REGION Network 2: Yeşil lamba
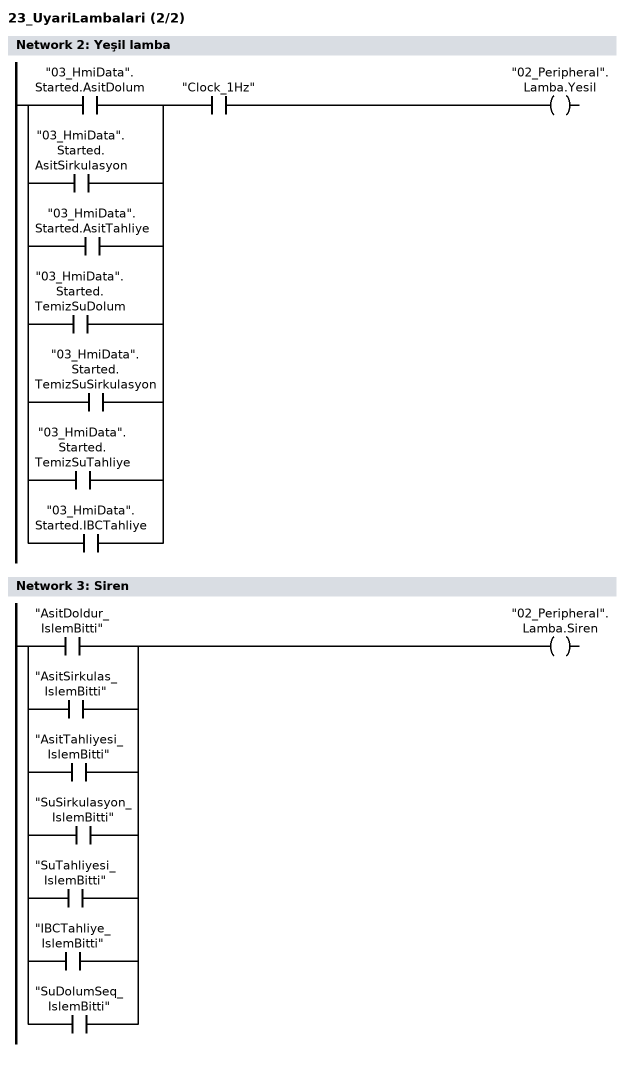
   RUNG wire#powerrail
      Contact( "03_HmiData".Started.AsitDolum )
      wire#w1
      Contact( "Clock_1Hz" )
      Coil( "02_Peripheral".Lamba.Yesil )
   END_RUNG
   RUNG wire#powerrail
      Contact( "03_HmiData".Started.AsitSirkulasyon )
   END_RUNG wire#w1
   RUNG wire#powerrail
      Contact( "03_HmiData".Started.AsitTahliye )
   END_RUNG wire#w1
   RUNG wire#powerrail
      Contact( "03_HmiData".Started.TemizSuDolum )
   END_RUNG wire#w1
   RUNG wire#powerrail
      Contact( "03_HmiData".Started.TemizSuSirkulasyon )
   END_RUNG wire#w1
   RUNG wire#powerrail
      Contact( "03_HmiData".Started.TemizSuTahliye )
   END_RUNG wire#w1
   RUNG wire#powerrail
      Contact( "03_HmiData".Started.IBCTahliye )
   END_RUNG wire#w1
   // the same network as SCL:
   "02_Peripheral".Lamba.Yesil := ("03_HmiData".Started.AsitDolum OR "03_HmiData".Started.AsitSirkulasyon OR "03_HmiData".Started.AsitTahliye OR "03_HmiData".Started.TemizSuDolum OR "03_HmiData".Started.TemizSuSirkulasyon OR "03_HmiData".Started.TemizSuTahliye OR "03_HmiData".Started.IBCTahliye) AND "Clock_1Hz";
END_REGION

REGION Network 3: Siren
   RUNG wire#powerrail
      Contact( "AsitDoldur_IslemBitti" )
      wire#w1
      Coil( "02_Peripheral".Lamba.Siren )
   END_RUNG
   RUNG wire#powerrail
      Contact( "AsitSirkulas_IslemBitti" )
   END_RUNG wire#w1
   RUNG wire#powerrail
      Contact( "AsitTahliyesi_IslemBitti" )
   END_RUNG wire#w1
   RUNG wire#powerrail
      Contact( "SuSirkulasyon_IslemBitti" )
   END_RUNG wire#w1
   RUNG wire#powerrail
      Contact( "SuTahliyesi_IslemBitti" )
   END_RUNG wire#w1
   RUNG wire#powerrail
      Contact( "IBCTahliye_IslemBitti" )
   END_RUNG wire#w1
   RUNG wire#powerrail
      Contact( "SuDolumSeq_IslemBitti" )
   END_RUNG wire#w1
   // the same network as SCL:
   "02_Peripheral".Lamba.Siren := "AsitDoldur_IslemBitti" OR "AsitSirkulas_IslemBitti" OR "AsitTahliyesi_IslemBitti" OR "SuSirkulasyon_IslemBitti" OR "SuTahliyesi_IslemBitti" OR "IBCTahliye_IslemBitti" OR "SuDolumSeq_IslemBitti";
END_REGION
END_FUNCTION

FUNCTION "14_SuDolumuSeq" : Void   // FC10, LAD
{ S7_Optimized_Access := 'TRUE' }
VERSION : 0.1
BEGIN

REGION Network 1
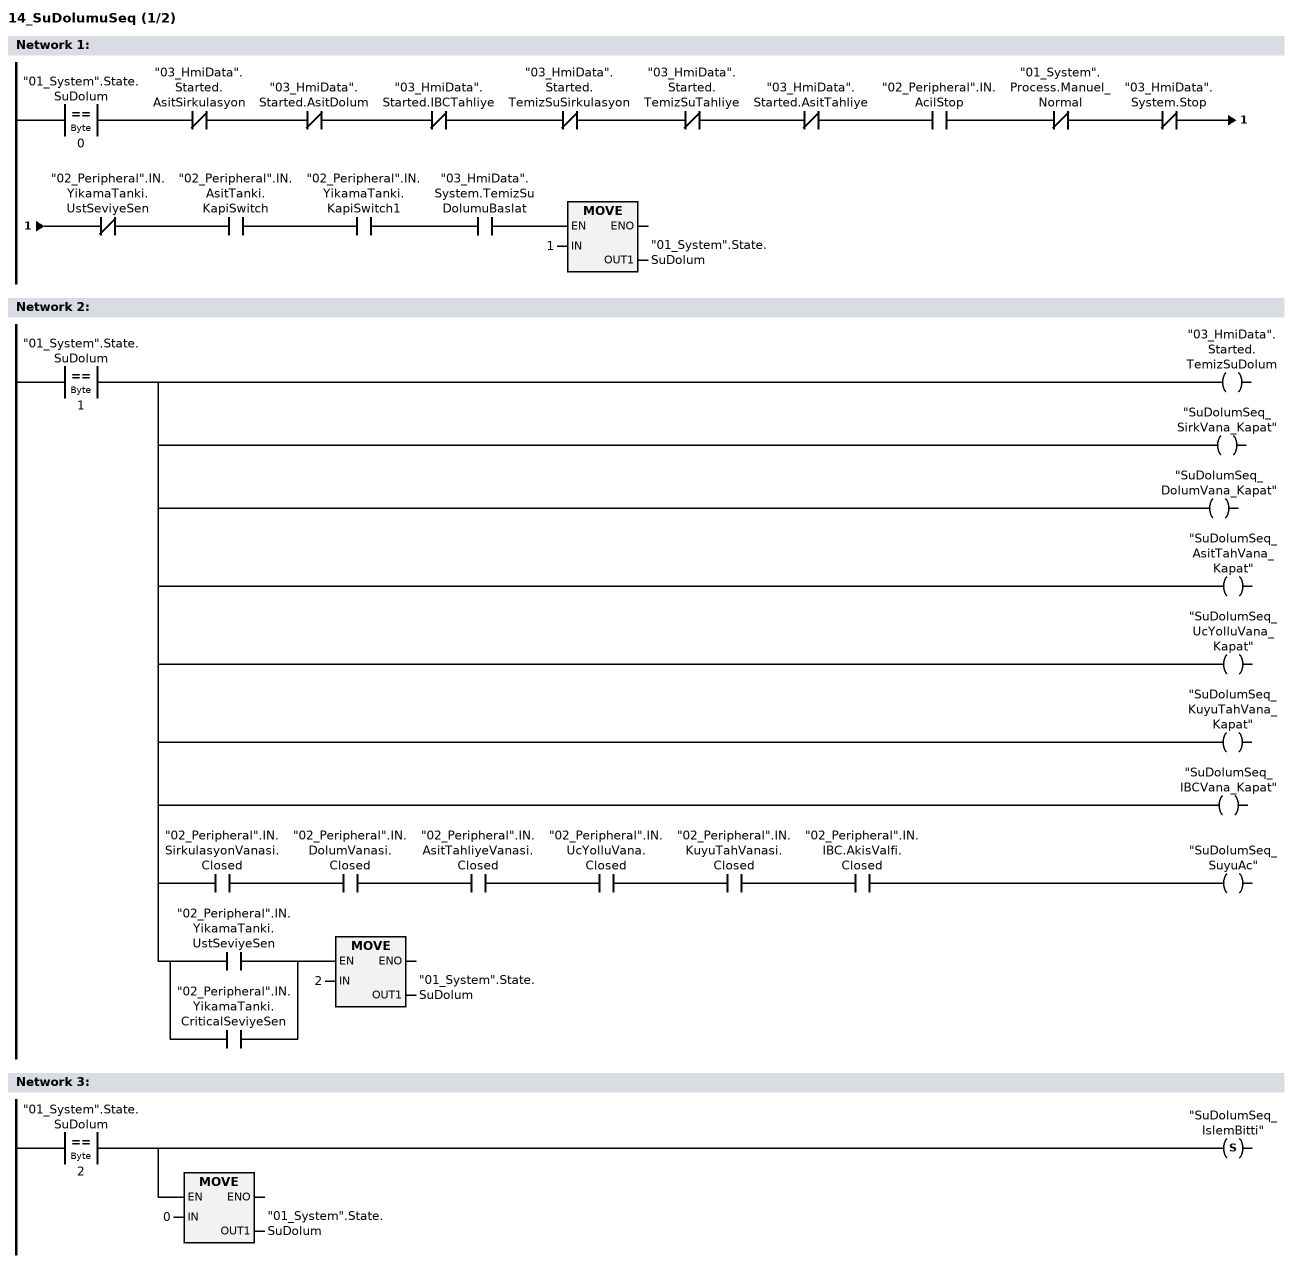
   RUNG wire#powerrail
      { S7_Templates := "SrcType := Byte" } EQ_Contact(in1 := "01_System".State.SuDolum, in2 := 0)
      I_Contact( "03_HmiData".Started.AsitSirkulasyon )
      I_Contact( "03_HmiData".Started.AsitDolum )
      I_Contact( "03_HmiData".Started.IBCTahliye )
      I_Contact( "03_HmiData".Started.TemizSuSirkulasyon )
      I_Contact( "03_HmiData".Started.TemizSuTahliye )
      I_Contact( "03_HmiData".Started.AsitTahliye )
      Contact( "02_Peripheral".IN.AcilStop )
      I_Contact( "01_System".Process.Manuel_Normal )
      I_Contact( "03_HmiData".System.Stop )
      I_Contact( "02_Peripheral".IN.YikamaTanki.UstSeviyeSen )
      Contact( "02_Peripheral".IN.AsitTanki.KapiSwitch )
      Contact( "02_Peripheral".IN.YikamaTanki.KapiSwitch1 )
      Contact( "03_HmiData".System.TemizSuDolumuBaslat )
      Move(in := 1, out1 => "01_System".State.SuDolum)
   END_RUNG
   // the same network as SCL:
   IF ("01_System".State.SuDolum = 0) AND NOT "03_HmiData".Started.AsitSirkulasyon AND NOT "03_HmiData".Started.AsitDolum AND NOT "03_HmiData".Started.IBCTahliye AND NOT "03_HmiData".Started.TemizSuSirkulasyon AND NOT "03_HmiData".Started.TemizSuTahliye AND NOT "03_HmiData".Started.AsitTahliye AND "02_Peripheral".IN.AcilStop AND NOT "01_System".Process.Manuel_Normal AND NOT "03_HmiData".System.Stop AND NOT "02_Peripheral".IN.YikamaTanki.UstSeviyeSen AND "02_Peripheral".IN.AsitTanki.KapiSwitch AND "02_Peripheral".IN.YikamaTanki.KapiSwitch1 AND "03_HmiData".System.TemizSuDolumuBaslat THEN
       "01_System".State.SuDolum := 1;
   END_IF;
END_REGION

REGION Network 2
   RUNG wire#powerrail
      { S7_Templates := "SrcType := Byte" } EQ_Contact(in1 := "01_System".State.SuDolum, in2 := 1)
      wire#w1
      Coil( "03_HmiData".Started.TemizSuDolum )
   END_RUNG
   RUNG wire#w1
      Coil( "SuDolumSeq_SirkVana_Kapat" )
   END_RUNG
   RUNG wire#w1
      Coil( "SuDolumSeq_DolumVana_Kapat" )
   END_RUNG
   RUNG wire#w1
      Coil( "SuDolumSeq_AsitTahVana_Kapat" )
   END_RUNG
   RUNG wire#w1
      Coil( "SuDolumSeq_UcYolluVana_Kapat" )
   END_RUNG
   RUNG wire#w1
      Coil( "SuDolumSeq_KuyuTahVana_Kapat" )
   END_RUNG
   RUNG wire#w1
      Coil( "SuDolumSeq_IBCVana_Kapat" )
   END_RUNG
   RUNG wire#w1
      Contact( "02_Peripheral".IN.SirkulasyonVanasi.Closed )
      Contact( "02_Peripheral".IN.DolumVanasi.Closed )
      Contact( "02_Peripheral".IN.AsitTahliyeVanasi.Closed )
      Contact( "02_Peripheral".IN.UcYolluVana.Closed )
      Contact( "02_Peripheral".IN.KuyuTahVanasi.Closed )
      Contact( "02_Peripheral".IN.IBC.AkisValfi.Closed )
      Coil( "SuDolumSeq_SuyuAc" )
   END_RUNG
   RUNG wire#w1
      Contact( "02_Peripheral".IN.YikamaTanki.UstSeviyeSen )
      wire#w2
      Move(in := 2, out1 => "01_System".State.SuDolum)
   END_RUNG
   RUNG wire#w1
      Contact( "02_Peripheral".IN.YikamaTanki.CriticalSeviyeSen )
   END_RUNG wire#w2
   // the same network as SCL:
   "03_HmiData".Started.TemizSuDolum := "01_System".State.SuDolum = 1;
   "SuDolumSeq_SirkVana_Kapat" := "03_HmiData".Started.TemizSuDolum;
   "SuDolumSeq_DolumVana_Kapat" := "03_HmiData".Started.TemizSuDolum;
   "SuDolumSeq_AsitTahVana_Kapat" := "03_HmiData".Started.TemizSuDolum;
   "SuDolumSeq_UcYolluVana_Kapat" := "03_HmiData".Started.TemizSuDolum;
   "SuDolumSeq_KuyuTahVana_Kapat" := "03_HmiData".Started.TemizSuDolum;
   "SuDolumSeq_IBCVana_Kapat" := "03_HmiData".Started.TemizSuDolum;
   "SuDolumSeq_SuyuAc" := "03_HmiData".Started.TemizSuDolum AND "02_Peripheral".IN.SirkulasyonVanasi.Closed AND "02_Peripheral".IN.DolumVanasi.Closed AND "02_Peripheral".IN.AsitTahliyeVanasi.Closed AND "02_Peripheral".IN.UcYolluVana.Closed AND "02_Peripheral".IN.KuyuTahVanasi.Closed AND "02_Peripheral".IN.IBC.AkisValfi.Closed;
   IF "03_HmiData".Started.TemizSuDolum AND ("02_Peripheral".IN.YikamaTanki.UstSeviyeSen OR "02_Peripheral".IN.YikamaTanki.CriticalSeviyeSen) THEN
       "01_System".State.SuDolum := 2;
   END_IF;
END_REGION

REGION Network 3
   RUNG wire#powerrail
      { S7_Templates := "SrcType := Byte" } EQ_Contact(in1 := "01_System".State.SuDolum, in2 := 2)
      wire#w1
      S_Coil( "SuDolumSeq_IslemBitti" )
   END_RUNG
   RUNG wire#w1
      Move(in := 0, out1 => "01_System".State.SuDolum)
   END_RUNG
   // the same network as SCL:
   IF "01_System".State.SuDolum = 2 THEN
       "SuDolumSeq_IslemBitti" := TRUE;
       "01_System".State.SuDolum := 0;
   END_IF;
END_REGION

REGION Network 4
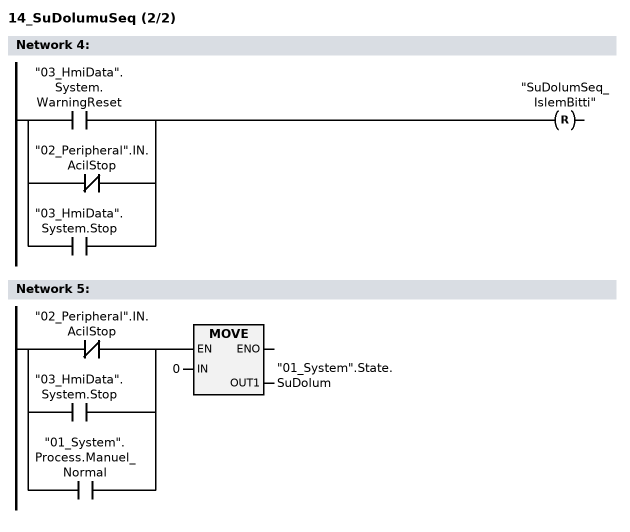
   RUNG wire#powerrail
      Contact( "03_HmiData".System.WarningReset )
      wire#w1
      R_Coil( "SuDolumSeq_IslemBitti" )
   END_RUNG
   RUNG wire#powerrail
      I_Contact( "02_Peripheral".IN.AcilStop )
   END_RUNG wire#w1
   RUNG wire#powerrail
      Contact( "03_HmiData".System.Stop )
   END_RUNG wire#w1
   // the same network as SCL:
   IF "03_HmiData".System.WarningReset OR NOT "02_Peripheral".IN.AcilStop OR "03_HmiData".System.Stop THEN
       "SuDolumSeq_IslemBitti" := FALSE;
   END_IF;
END_REGION

REGION Network 5
   RUNG wire#powerrail
      I_Contact( "02_Peripheral".IN.AcilStop )
      wire#w1
      Move(in := 0, out1 => "01_System".State.SuDolum)
   END_RUNG
   RUNG wire#powerrail
      Contact( "03_HmiData".System.Stop )
   END_RUNG wire#w1
   RUNG wire#powerrail
      Contact( "01_System".Process.Manuel_Normal )
   END_RUNG wire#w1
   // the same network as SCL:
   IF NOT "02_Peripheral".IN.AcilStop OR "03_HmiData".System.Stop OR "01_System".Process.Manuel_Normal THEN
       "01_System".State.SuDolum := 0;
   END_IF;
END_REGION
END_FUNCTION

ORGANIZATION_BLOCK "Main"   // OB1, FBD, ProgramCycle
TITLE = "Main Program Sweep (Cycle)"
{ S7_Optimized_Access := 'TRUE' }
VERSION : 0.1
   VAR_INPUT
      Initial_Call : Bool;   // Initial call of this OB
      Remanence : Bool;   // =True, if remanent data are available
   END_VAR
BEGIN

REGION Network 1: Manuel
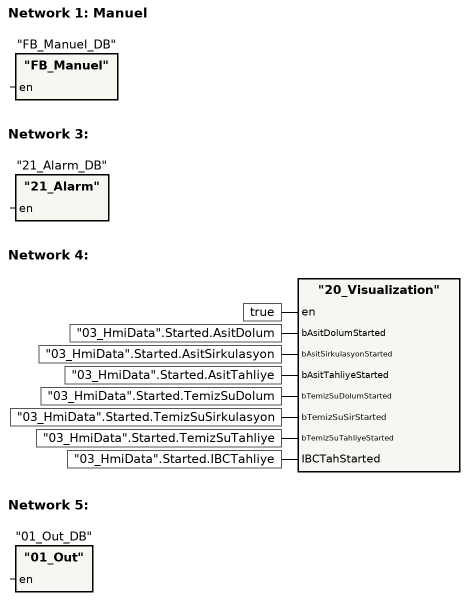
   "FB_Manuel_DB"();   // "FB_Manuel"
END_REGION

REGION Network 2 (SCL): Otomatik sekanslar
   "11_AsitDolumSeq"();
   "12_AsitSirkulasyonSeq"();
   "13_AsitTahliyeSeq"();
   "14_SuDolumuSeq"();
   "15_SuSirkulasyonSeq"();
   "16_SuTahliyeSeq"();
   "17_IBCTahliyeSeq"();

   "22_Peripheral"();
   "23_UyariLambalari"();

   "Always_On" := true;
END_REGION

REGION Network 3
   "21_Alarm_DB"();   // "21_Alarm"
END_REGION

REGION Network 4
   IF true THEN
       "20_Visualization"(bAsitDolumStarted := "03_HmiData".Started.AsitDolum,
                          bAsitSirkulasyonStarted := "03_HmiData".Started.AsitSirkulasyon,
                          bAsitTahliyeStarted := "03_HmiData".Started.AsitTahliye,
                          bTemizSuDolumStarted := "03_HmiData".Started.TemizSuDolum,
                          bTemizSuSirStarted := "03_HmiData".Started.TemizSuSirkulasyon,
                          bTemizSuTahliyeStarted := "03_HmiData".Started.TemizSuTahliye,
                          IBCTahStarted := "03_HmiData".Started.IBCTahliye);
   END_IF;
END_REGION

REGION Network 5
   "01_Out_DB"();   // "01_Out"
END_REGION
END_ORGANIZATION_BLOCK

// folder: OB

ORGANIZATION_BLOCK "Time error interrupt"   // OB80, LAD, TimeErrorInterrupt
{ S7_Optimized_Access := 'TRUE' }
VERSION : 0.1
   VAR_INPUT
      Fault_ID : Byte;   // Fault identifier
      Csg_OBnr : OB_Any;   // Number of OB causing the error
      Csg_Prio : UInt;   // Priority of OB causing the error
   END_VAR
BEGIN
END_ORGANIZATION_BLOCK

ORGANIZATION_BLOCK "Pull or plug of modules"   // OB83, LAD, PullPlug
{ S7_Optimized_Access := 'TRUE' }
VERSION : 0.1
   VAR_INPUT
      LADDR : Hw_Io;   // Hardware identifier
      Event_Class : Byte;   // 16#38/39: module inserted, removed
      Fault_ID : Byte;   // Fault identifier
   END_VAR
BEGIN
END_ORGANIZATION_BLOCK

ORGANIZATION_BLOCK "Rack or station failure"   // OB86, LAD, RackStationFailure
{ S7_Optimized_Access := 'TRUE' }
VERSION : 0.1
   VAR_INPUT
      LADDR : Hw_Device;   // Hardware identifier
      Event_Class : Byte;   // Event class
      Fault_ID : Byte;   // Fault identifier
   END_VAR
BEGIN
END_ORGANIZATION_BLOCK

ORGANIZATION_BLOCK "Startup"   // OB100, LAD, Startup
TITLE = "Complete Restart"
{ S7_Optimized_Access := 'TRUE' }
VERSION : 0.1
   VAR_INPUT
      LostRetentive : Bool;   // True if retentive data are lost
      LostRTC : Bool;   // True if date and time are lost
   END_VAR
BEGIN

REGION Network 1
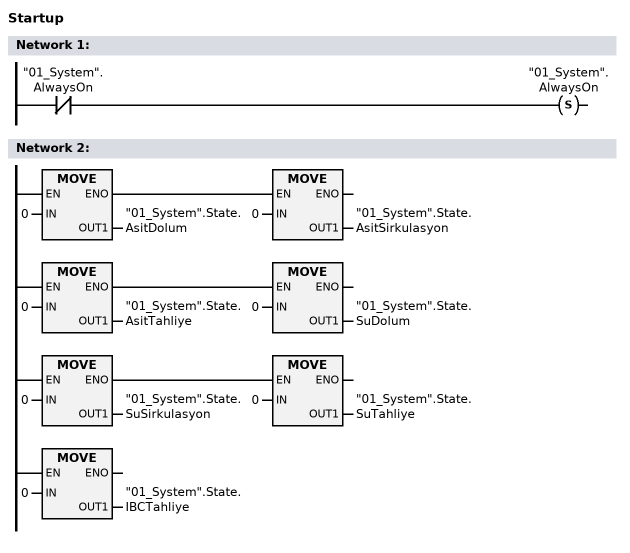
   RUNG wire#powerrail
      I_Contact( "01_System".AlwaysOn )
      S_Coil( "01_System".AlwaysOn )
   END_RUNG
   // the same network as SCL:
   IF NOT "01_System".AlwaysOn THEN "01_System".AlwaysOn := TRUE; END_IF;
END_REGION

REGION Network 2
   RUNG wire#powerrail
      Move(in := 0, out1 => "01_System".State.AsitDolum)
      Move(in := 0, out1 => "01_System".State.AsitSirkulasyon)
   END_RUNG
   RUNG wire#powerrail
      Move(in := 0, out1 => "01_System".State.AsitTahliye)
      Move(in := 0, out1 => "01_System".State.SuDolum)
   END_RUNG
   RUNG wire#powerrail
      Move(in := 0, out1 => "01_System".State.SuSirkulasyon)
      Move(in := 0, out1 => "01_System".State.SuTahliye)
   END_RUNG
   RUNG wire#powerrail
      Move(in := 0, out1 => "01_System".State.IBCTahliye)
   END_RUNG
   // the same network as SCL:
   "01_System".State.AsitDolum := 0;
   "01_System".State.AsitSirkulasyon := 0;
   "01_System".State.AsitTahliye := 0;
   "01_System".State.SuDolum := 0;
   "01_System".State.SuSirkulasyon := 0;
   "01_System".State.SuTahliye := 0;
   "01_System".State.IBCTahliye := 0;
END_REGION
END_ORGANIZATION_BLOCK

(* ===== HMI "HMI_RT_1" =====
system functions are stored by id; their names below are inferred from use
connection "HMI_Connection_1": ETHERNET, SMART_S7_1200_OMS

HMI tags "Default tag table"
   "01_System_SystemInfo" : String[50] = PLC "01_System".SystemInfo, 100 ms
   "TestInfo" : WString[254] AT %DB1.DBX0.0
   "01_System_Alarms" : Word = PLC "01_System".Alarms, 1 s
   "01_System_Process.Manuel_Normal" : Bool = PLC "01_System".Process.Manuel_Normal, 100 ms
   "02_Peripheral_OUT.KorKuyuPompasi" : Bool = PLC "02_Peripheral".OUT.KorKuyuPompasi, 500 ms
   "HmiAnaPompa_Run" : Bool = PLC HmiAnaPompa_Run AT %M2.4, 1 s
   "HmiIBCPopmpa_Run" : Bool = PLC HmiIBCPopmpa_Run AT %M2.5, 1 s
   "HmiKorKuyuPompa_Run" : Bool = PLC HmiKorKuyuPompa_Run AT %M10.5, 1 s
   "03_HmiData_SoDulumVanasi_Ac" : Bool = PLC "03_HmiData".SuDolumVanasi_Ac, 1 s
   "03_HmiData_SuDolumVanasi_Kapat" : Bool = PLC "03_HmiData".SuDolumVanasi_Kapat, 1 s
   "02_Peripheral_OUT.SuDolumVanasi" : Bool = PLC "02_Peripheral".OUT.SuDolumVanasi, 1 s

HMI tags "00_HMI"
   "03_HmiData_SurkilasyonVanasi_Ac" : Bool = PLC "03_HmiData".SurkilasyonVanasi_Ac, 100 ms
   "03_HmiData_SurkilasyonVanasi_Kapat" : Bool = PLC "03_HmiData".SurkilasyonVanasi_Kapat, 100 ms
   "03_HmiData_DolumVanasi_Ac" : Bool = PLC "03_HmiData".DolumVanasi_Ac, 100 ms
   "03_HmiData_DolumVanasi_Kapat" : Bool = PLC "03_HmiData".DolumVanasi_Kapat, 100 ms
   "03_HmiData_AsitTahliyeVanasi_Ac" : Bool = PLC "03_HmiData".AsitTahliyeVanasi_Ac, 100 ms
   "03_HmiData_AsitTahliyeVanasi_Kapat" : Bool = PLC "03_HmiData".AsitTahliyeVanasi_Kapat, 100 ms
   "03_HmiData_UcYolluVana_Ac" : Bool = PLC "03_HmiData".UcYolluVana_Ac, 100 ms
   "03_HmiData_UcYolluVana_Kapat" : Bool = PLC "03_HmiData".UcYolluVana_Kapat, 100 ms
   "03_HmiData_KuyuAktarimVanasi_Ac" : Bool = PLC "03_HmiData".KuyuAktarimVanasi_Ac, 100 ms
   "03_HmiData_KuyuAktarimVanasi_Kapat" : Bool = PLC "03_HmiData".KuyuAktarimVanasi_Kapat, 100 ms
   "03_HmiData_IBCVanasi_Ac" : Bool = PLC "03_HmiData".IBCVanasi_Ac, 100 ms
   "03_HmiData_IBCVanasi_Kapat" : Bool = PLC "03_HmiData".IBCVanasi_Kapat, 100 ms
   "03_HmiData_AnaPompa_Run" : Bool = PLC "03_HmiData".AnaPompa_Run, 100 ms
   "03_HmiData_AnaPompa_Stop" : Bool = PLC "03_HmiData".AnaPompa_Stop, 100 ms
   "03_HmiData_IBC_DiyaframPompa_Run" : Bool = PLC "03_HmiData".IBC_DiyaframPompa_Run, 100 ms
   "03_HmiData_IBC_DiyaframPompa_Stop" : Bool = PLC "03_HmiData".IBC_DiyaframPompa_Stop, 100 ms
   "03_HmiData_Started.AsitDolum" : Bool = PLC "03_HmiData".Started.AsitDolum, 1 s
   "03_HmiData_Started.AsitSirkulasyon" : Bool = PLC "03_HmiData".Started.AsitSirkulasyon, 1 s
   "03_HmiData_Started.AsitTahliye" : Bool = PLC "03_HmiData".Started.AsitTahliye, 1 s
   "03_HmiData_Started.IBCTahliye" : Bool = PLC "03_HmiData".Started.IBCTahliye, 1 s
   "03_HmiData_Started.TemizSuDolum" : Bool = PLC "03_HmiData".Started.TemizSuDolum, 1 s
   "03_HmiData_Started.TemizSuSirkulasyon" : Bool = PLC "03_HmiData".Started.TemizSuSirkulasyon, 1 s
   "03_HmiData_Started.TemizSuTahliye" : Bool = PLC "03_HmiData".Started.TemizSuTahliye, 1 s
   "03_HmiData_System.Stop" : Bool = PLC "03_HmiData".System.Stop, 1 s
   "03_HmiData_System.WarningReset" : Bool = PLC "03_HmiData".System.WarningReset, 1 s
   "03_HmiData_Visualization.ActTimer" : DInt = PLC "03_HmiData".Visualization.ActTimerMin, 1 s
   "03_HmiData_Visualization.TimerVisible" : Bool = PLC "03_HmiData".Visualization.TimerVisible, 1 s
   "03_HmiData_Visualization.Visibility.AsitDolum" : Bool = PLC "03_HmiData".Visualization.Visibility.AsitDolum, 1 s
   "03_HmiData_Visualization.Visibility.AsitSirkulasyon" : Bool = PLC "03_HmiData".Visualization.Visibility.AsitSirkulasyon, 1 s
   "03_HmiData_Visualization.Visibility.AsitTahliyesi" : Bool = PLC "03_HmiData".Visualization.Visibility.AsitTahliyesi, 1 s
   "03_HmiData_Visualization.Visibility.IBCTaliye" : Bool = PLC "03_HmiData".Visualization.Visibility.IBCTaliye, 1 s
   "03_HmiData_Visualization.Visibility.TemizSuDolum" : Bool = PLC "03_HmiData".Visualization.Visibility.TemizSuDolum, 1 s
   "03_HmiData_Visualization.Visibility.TemizSuSirkulasyon" : Bool = PLC "03_HmiData".Visualization.Visibility.TemizSuSirkulasyon, 1 s
   "03_HmiData_Visualization.Visibility.TemizSuTahliye" : Bool = PLC "03_HmiData".Visualization.Visibility.TemizSuTahliye, 1 s
   "03_HmiData_KorKuyuPompası_Run" : Bool = PLC "03_HmiData".KorKuyuPompası_Run, 500 ms
   "03_HmiData_KorKuyuPompası_Stop" : Bool = PLC "03_HmiData".KorKuyuPompası_Stop, 500 ms
   "03_HmiData_System.AsitDoldurBaslat" : Bool = PLC "03_HmiData".System.AsitDoldurBaslat, 500 ms
   "03_HmiData_System.AsitSirkulasyonBaslat" : Bool = PLC "03_HmiData".System.AsitSirkulasyonBaslat, 500 ms
   "03_HmiData_System.AsitTahliyesiBaslat" : Bool = PLC "03_HmiData".System.AsitTahliyesiBaslat, 500 ms
   "03_HmiData_System.IBCTahliyesiBaslat" : Bool = PLC "03_HmiData".System.IBCTahliyesiBaslat, 500 ms
   "03_HmiData_System.TemizSuDolumuBaslat" : Bool = PLC "03_HmiData".System.TemizSuDolumuBaslat, 500 ms
   "03_HmiData_System.TemizSuSirkulasyonuBaslat" : Bool = PLC "03_HmiData".System.TemizSuSirkulasyonuBaslat, 500 ms
   "03_HmiData_System.TemizSuTahliyesiBaslat" : Bool = PLC "03_HmiData".System.TemizSuTahliyesiBaslat, 500 ms
   "03_HmiData_TimerInterval.AsitSirkulasyon" : Time = PLC "03_HmiData".TimerInterval.AsitSirkulasyon, 500 ms
   "03_HmiData_TimerInterval.SuSirkulasyon" : Time = PLC "03_HmiData".TimerInterval.SuSirkulasyon, 500 ms
   "03_HmiData_Visualization.ActTimerSec" : DInt = PLC "03_HmiData".Visualization.ActTimerSec, 100 ms
   "03_HmiData_Visualization.Visibility.Manuel.AsitTahVanaAc" : Bool = PLC "03_HmiData".Visualization.Visibility.Manuel.AsitTahVanaAc, 1 s
   "03_HmiData_Visualization.Visibility.Manuel.AsitTahVanaKapat" : Bool = PLC "03_HmiData".Visualization.Visibility.Manuel.AsitTahVanaKapat, 1 s
   "03_HmiData_Visualization.Visibility.Manuel.DolumVanaAc" : Bool = PLC "03_HmiData".Visualization.Visibility.Manuel.DolumVanaAc, 1 s
   "03_HmiData_Visualization.Visibility.Manuel.DolumVanaKapat" : Bool = PLC "03_HmiData".Visualization.Visibility.Manuel.DolumVanaKapat, 1 s
   "03_HmiData_Visualization.Visibility.Manuel.IBCVanaAc" : Bool = PLC "03_HmiData".Visualization.Visibility.Manuel.IBCVanaAc, 1 s
   "03_HmiData_Visualization.Visibility.Manuel.IBCVanaKapat" : Bool = PLC "03_HmiData".Visualization.Visibility.Manuel.IBCVanaKapat, 1 s
   "03_HmiData_Visualization.Visibility.Manuel.KuyuTahVanaAc" : Bool = PLC "03_HmiData".Visualization.Visibility.Manuel.KuyuTahVanaAc, 1 s
   "03_HmiData_Visualization.Visibility.Manuel.KuyuTahVanaKapat" : Bool = PLC "03_HmiData".Visualization.Visibility.Manuel.KuyuTahVanaKapat, 1 s
   "03_HmiData_Visualization.Visibility.Manuel.SirkulasyonVanaAc" : Bool = PLC "03_HmiData".Visualization.Visibility.Manuel.SirkulasyonVanaAc, 1 s
   "03_HmiData_Visualization.Visibility.Manuel.SirkulasyonVanaKapat" : Bool = PLC "03_HmiData".Visualization.Visibility.Manuel.SirkulasyonVanaKapat, 1 s
   "03_HmiData_Visualization.Visibility.Manuel.UcYolluVanaAc" : Bool = PLC "03_HmiData".Visualization.Visibility.Manuel.UcYolluVanaAc, 1 s
   "03_HmiData_Visualization.Visibility.Manuel.UcYolluVanaKapat" : Bool = PLC "03_HmiData".Visualization.Visibility.Manuel.UcYolluVanaKapat, 1 s

HMI tags "01_Peripheral"
   "02_Peripheral_IN.AsitTahliyeVanasi.Closed" : Bool = PLC "02_Peripheral".IN.AsitTahliyeVanasi.Closed, 500 ms
   "02_Peripheral_IN.AsitTahliyeVanasi.Opened" : Bool = PLC "02_Peripheral".IN.AsitTahliyeVanasi.Opened, 500 ms
   "02_Peripheral_IN.DolumVanasi.Closed" : Bool = PLC "02_Peripheral".IN.DolumVanasi.Closed, 500 ms
   "02_Peripheral_IN.DolumVanasi.Opened" : Bool = PLC "02_Peripheral".IN.DolumVanasi.Opened, 500 ms
   "02_Peripheral_IN.IBC.AkisValfi.Closed" : Bool = PLC "02_Peripheral".IN.IBC.AkisValfi.Closed, 500 ms
   "02_Peripheral_IN.IBC.AkisValfi.Opened" : Bool = PLC "02_Peripheral".IN.IBC.AkisValfi.Opened, 500 ms
   "02_Peripheral_IN.KuyuAktVanasi.Closed" : Bool = PLC "02_Peripheral".IN.KuyuTahVanasi.Closed, 500 ms
   "02_Peripheral_IN.KuyuAktVanasi.Opened" : Bool = PLC "02_Peripheral".IN.KuyuTahVanasi.Opened, 500 ms
   "02_Peripheral_IN.SirkulasyonVanasi.Closed" : Bool = PLC "02_Peripheral".IN.SirkulasyonVanasi.Closed, 500 ms
   "02_Peripheral_IN.SirkulasyonVanasi.Opened" : Bool = PLC "02_Peripheral".IN.SirkulasyonVanasi.Opened, 500 ms
   "02_Peripheral_IN.UcYolluVana.Closed" : Bool = PLC "02_Peripheral".IN.UcYolluVana.Closed, 500 ms
   "02_Peripheral_IN.UcYolluVana.Opened" : Bool = PLC "02_Peripheral".IN.UcYolluVana.Opened, 500 ms
   "02_Peripheral_OUT.AnaPompa" : Bool = PLC "02_Peripheral".OUT.AnaPompa, 500 ms
   "02_Peripheral_OUT.IBC.PompaDiyafram" : Bool = PLC "02_Peripheral".OUT.IBC.PompaDiyafram, 500 ms
   "02_Peripheral_IN.AsitTanki.AltSeviyeSen" : Bool = PLC "02_Peripheral".IN.AsitTanki.AltSeviyeSen, 1 s
   "02_Peripheral_IN.AsitTanki.KapiSwitch" : Bool = PLC "02_Peripheral".IN.AsitTanki.KapiSwitch, 500 ms
   "02_Peripheral_IN.AsitTanki.UstSeviyeSen" : Bool = PLC "02_Peripheral".IN.AsitTanki.UstSeviyeSen, 1 s
   "02_Peripheral_IN.YikamaTanki.AltSeviyeSen" : Bool = PLC "02_Peripheral".IN.YikamaTanki.AltSeviyeSen, 1 s
   "02_Peripheral_IN.YikamaTanki.KapiSwitch1" : Bool = PLC "02_Peripheral".IN.YikamaTanki.KapiSwitch1, 500 ms
   "02_Peripheral_IN.YikamaTanki.KapiSwitch2" : Bool = PLC "02_Peripheral".IN.YikamaTanki.KapiSwitch2, 500 ms
   "02_Peripheral_IN.YikamaTanki.UstSeviyeSen" : Bool = PLC "02_Peripheral".IN.YikamaTanki.UstSeviyeSen, 1 s

discrete alarms
   1: 'Acil stop basılı', class Errors, trigger "01_System_Alarms" bit 0
   2: 'Ana pompa termik hatası', class Errors, trigger "01_System_Alarms" bit 1
   3: 'Sirkulasyon vanası açılma sorunu', class Errors, trigger "01_System_Alarms" bit 2
   4: 'Sirkulasyon vanası kapanma sorunu', class Errors, trigger "01_System_Alarms" bit 3
   5: 'Dolum vanası açılma sorunu', class Errors, trigger "01_System_Alarms" bit 4
   6: 'Dolum vanası kapanma sorunu', class Errors, trigger "01_System_Alarms" bit 5
   7: 'Asit tahliye vanası açılma sorunu', class Errors, trigger "01_System_Alarms" bit 6
   8: 'Asit tahliye vanası kapanma sorunu', class Errors, trigger "01_System_Alarms" bit 7
   9: 'Üç yollu vana açılma sorunu', class Errors, trigger "01_System_Alarms" bit 8
   10: 'Üç yollu vana kapanma sorunu', class Errors, trigger "01_System_Alarms" bit 9
   11: 'Kuyu tahliye vanası açılma sorunu', class Errors, trigger "01_System_Alarms" bit 10
   12: 'Kuyu tahliye vanası kapanma sorunu', class Errors, trigger "01_System_Alarms" bit 11
   13: 'IBC tahliye vanası açılma sorunu', class Errors, trigger "01_System_Alarms" bit 12
   14: 'IBC tahliye vanası kapanma sorunu', class Errors, trigger "01_System_Alarms" bit 13
   15: 'Yıkama tankı kritik seviyede', class Errors, trigger "01_System_Alarms" bit 14
   16: 'Asit tankında yeterli asit yok', class Errors, trigger "01_System_Alarms" bit 15

Template "00_RootTamplate" 480x272
   Button "Template_Button" at 293,223 size 88x44; TextOff 'İzleme'
      on Release: ActivateScreen("03_Izleme", 0)
   Button "Template_Button_1" at 195,223 size 88x44; TextOff 'Manuel'
      on Release: ActivateScreen("01_Manuel", 0)
   Button "Alarms" at 99,223 size 88x44; TextOff 'Alarm'; TextOn 'Alarms'; PictureOff "AlarmDisplay_KTP400_Basic_color_PN"; PictureOn "AlarmDisplay_KTP400_Basic_color_PN"
      on Release: ActivateScreen("02_Alarm", 0)
   Button "Start screen" at 4,223 size 88x44; TextOff 'Ana Ekran'; TextOn 'Start screen'; PictureOff "NavigateHome_KTP400_Basic_color_PN"; PictureOn "NavigateHome_KTP400_Basic_color_PN"
      on Release: ActivateScreen("00_Root screen", 0)
   Button "Template_Button_2" at 388,223 size 88x44; TextOff 'Süreler'
      on Release: ActivateScreen("04_Sure", 0)

screen "00_Root screen" 480x272, template "00_RootTamplate"
   IOField "Template_I/O field_1" at 6,2 size 351x44; FormatPattern ??????????????????????????????????????????????????
      ProcessValue <- "01_System_SystemInfo"
   Button "Button_9" at 5,54 size 169x49; TextOff 'NORMAL'; TextOn 'MANUEL'; TextList "TextList_Manuel_Normal"
      on Release: InvertBit("01_System_Process.Manuel_Normal")
      Appearance <- "01_System_Process.Manuel_Normal"
      ProcessValue <- "01_System_Process.Manuel_Normal"
   Rectangle "Rectangle_1" at 358,1 size 121x47
      Visibility <- "03_HmiData_Visualization.TimerVisible"
   IOField "I/O field_3" at 361,21 size 69x24; FormatPattern 99999; Unit  dk
      ProcessValue <- "03_HmiData_Visualization.ActTimer"
      Visibility <- "03_HmiData_Visualization.TimerVisible"
   TextField "Text field_3" at 380,1 size 80x18; Text 'Geçen Sure:'
      Visibility <- "03_HmiData_Visualization.TimerVisible"
   IOField "I/O field_4" at 430,21 size 46x24; FormatPattern 99; Unit  sn
      Visibility <- "03_HmiData_Visualization.TimerVisible"
      ProcessValue <- "03_HmiData_Visualization.ActTimerSec"
   Button "Button_15" at 186,54 size 136x49; TextOff 'Asit Doldur Başlat'
      on Press: function_b14e0dd5("03_HmiData_System.AsitDoldurBaslat", 0)
      Appearance <- "03_HmiData_Started.AsitDolum"
   Button "Button_1" at 186,113 size 136x50; TextOff 'Asit Sirkülasyon Başlat'
      on Press: function_b14e0dd5("03_HmiData_System.AsitSirkulasyonBaslat", 0)
      Appearance <- "03_HmiData_Started.AsitSirkulasyon"
   Button "Button_2" at 186,167 size 136x50; TextOff 'Asit Tahliyesi Başlat'
      on Press: function_b14e0dd5("03_HmiData_System.AsitTahliyesiBaslat", 0)
      Appearance <- "03_HmiData_Started.AsitTahliye"
   Button "Button_4" at 336,113 size 135x50; TextOff 'Su Sirkülasyon Başlat'
      on Press: function_b14e0dd5("03_HmiData_System.TemizSuSirkulasyonuBaslat", 0)
      Appearance <- "03_HmiData_Started.TemizSuSirkulasyon"
   Button "Button_5" at 336,167 size 135x50; TextOff 'Su Tahliyesi Başlat'
      on Press: function_b14e0dd5("03_HmiData_System.TemizSuTahliyesiBaslat", 0)
      Appearance <- "03_HmiData_Started.TemizSuTahliye"
   Button "Button_6" at 6,168 size 169x49; TextOff 'IBC Tahliye Başlat'
      on Press: function_b14e0dd5("03_HmiData_System.IBCTahliyesiBaslat", 0)
      Appearance <- "03_HmiData_Started.IBCTahliye"
   Button "Button_7" at 6,113 size 83x49; TextOff 'Uyarı Sustur'
      on Press: function_b14e0dd5("03_HmiData_System.WarningReset", 0)
   Button "Button_8" at 92,113 size 83x49; TextOff 'İşlemi Durdur'
      on Press: function_b14e0dd5("03_HmiData_System.Stop", 0)
   Button "Button_3" at 336,54 size 135x49; TextOff 'Su Doldur Başlat'
      on Press: function_b14e0dd5("03_HmiData_System.TemizSuDolumuBaslat", 0)
      Appearance <- "03_HmiData_Started.TemizSuDolum"

screen "01_Manuel" 480x272, template "00_RootTamplate"
   Button "Button_1" at 4,27 size 74x39; TextOff 'Ac'
      on Release: InvertBit("03_HmiData_SurkilasyonVanasi_Ac")
      Appearance <- "03_HmiData_SurkilasyonVanasi_Ac"
   Button "Button_2" at 4,97 size 74x39; TextOff 'Ac'
      on Release: InvertBit("03_HmiData_DolumVanasi_Ac")
      Visibility <- "03_HmiData_Visualization.Visibility.Manuel.DolumVanaAc"
      Appearance <- "03_HmiData_DolumVanasi_Ac"
   Button "Button_3" at 173,27 size 74x39; TextOff 'Ac'
      on Release: InvertBit("03_HmiData_UcYolluVana_Ac")
      Visibility <- "03_HmiData_Visualization.Visibility.Manuel.UcYolluVanaAc"
      Appearance <- "03_HmiData_UcYolluVana_Ac"
   Button "Button_5" at 173,97 size 74x39; TextOff 'Ac'
      on Release: InvertBit("03_HmiData_KuyuAktarimVanasi_Ac")
      Visibility <- "03_HmiData_Visualization.Visibility.Manuel.KuyuTahVanaAc"
      Appearance <- "03_HmiData_KuyuAktarimVanasi_Ac"
   Button "Button_4" at 4,171 size 74x39; TextOff 'Ac'
      on Release: InvertBit("03_HmiData_AsitTahliyeVanasi_Ac")
      Visibility <- "03_HmiData_Visualization.Visibility.Manuel.AsitTahVanaAc"
      Appearance <- "03_HmiData_AsitTahliyeVanasi_Ac"
   Button "Button_6" at 173,171 size 74x39; TextOff 'Ac'
      on Release: InvertBit("03_HmiData_IBCVanasi_Ac")
      Visibility <- "03_HmiData_Visualization.Visibility.Manuel.IBCVanaAc"
      Appearance <- "03_HmiData_IBCVanasi_Ac"
   Button "Button_9" at 88,27 size 74x39; TextOff 'Kapat'
      on Release: InvertBit("03_HmiData_SurkilasyonVanasi_Kapat")
      Appearance <- "03_HmiData_SurkilasyonVanasi_Kapat"
   Button "Button_10" at 254,27 size 74x39; TextOff 'Kapat'
      on Release: InvertBit("03_HmiData_UcYolluVana_Kapat")
      Visibility <- "03_HmiData_Visualization.Visibility.Manuel.UcYolluVanaKapat"
      Appearance <- "03_HmiData_UcYolluVana_Kapat"
   Button "Button_11" at 87,97 size 74x39; TextOff 'Kapat'
      on Release: InvertBit("03_HmiData_DolumVanasi_Kapat")
      Visibility <- "03_HmiData_Visualization.Visibility.Manuel.DolumVanaKapat"
      Appearance <- "03_HmiData_DolumVanasi_Kapat"
   Button "Button_12" at 87,171 size 74x39; TextOff 'Kapat'
      on Release: InvertBit("03_HmiData_AsitTahliyeVanasi_Kapat")
      Visibility <- "03_HmiData_Visualization.Visibility.Manuel.AsitTahVanaKapat"
      Appearance <- "03_HmiData_AsitTahliyeVanasi_Kapat"
   Button "Button_13" at 255,97 size 74x39; TextOff 'Kapat'
      on Release: InvertBit("03_HmiData_KuyuAktarimVanasi_Kapat")
      Visibility <- "03_HmiData_Visualization.Visibility.Manuel.KuyuTahVanaKapat"
      Appearance <- "03_HmiData_KuyuAktarimVanasi_Kapat"
   Button "Button_14" at 254,171 size 74x39; TextOff 'Kapat'
      on Release: InvertBit("03_HmiData_IBCVanasi_Kapat")
      Visibility <- "03_HmiData_Visualization.Visibility.Manuel.IBCVanaKapat"
      Appearance <- "03_HmiData_IBCVanasi_Kapat"
   Button "Button_7" at 357,26 size 102x39; TextOff 'Ac'
      Visibility <- "03_HmiData_Visualization.Visibility.Manuel.IBCVanaAc"
      Appearance <- "03_HmiData_SoDulumVanasi_Ac"
      on Press: function_b14e0dd5("03_HmiData_SoDulumVanasi_Ac", 0)
   Button "Button_8" at 357,67 size 102x39; TextOff 'Kapat'
      Visibility <- "03_HmiData_Visualization.Visibility.Manuel.IBCVanaKapat"
      Appearance <- "03_HmiData_SuDolumVanasi_Kapat"
      on Press: function_b14e0dd5("03_HmiData_SuDolumVanasi_Kapat", 0)
   TextField "Text field_1" at 25,5 size 123x18; Text 'Sirkülasyon Vanasi'
   TextField "Text field_3" at 31,78 size 118x18; Text 'Asit Dolum Vanasi'
   TextField "Text field_4" at 21,149 size 124x18; Text 'Asit Tahliye Vanasi'
   TextField "Text field_5" at 214,5 size 89x18; Text 'Uc Yollu Vana'
   TextField "Text field_6" at 185,78 size 136x18; Text 'Kuyu Aktarım Vanası'
   TextField "Text field_7" at 216,150 size 70x18; Text 'IBC Vanasi'
   TextField "Text field_2" at 353,6 size 108x18; Text 'Su Dolum Vanası'
   Button "Button_15" at 364,168 size 86x43; TextOff 'Text'; PictureOff "Right_Arrow"
      on Release: ActivateScreen("01_Manuel_Syf2", 0)
   TextField "Text field_8" at 353,6 size 108x18; Text 'Su Dolum Vanası'
   TextField "Text field_9" at 381,145 size 51x18; Text 'Sayfa 2'
   Rectangle "Rectangle_9" at 78,27 size 6x39
      Appearance <- "02_Peripheral_IN.SirkulasyonVanasi.Opened"
   Rectangle "Rectangle_10" at 161,27 size 6x39
      Appearance <- "02_Peripheral_IN.SirkulasyonVanasi.Closed"
   Rectangle "Rectangle_11" at 78,97 size 6x39
      Appearance <- "02_Peripheral_IN.DolumVanasi.Opened"
   Rectangle "Rectangle_12" at 161,97 size 6x39
      Appearance <- "02_Peripheral_IN.DolumVanasi.Closed"
   Rectangle "Rectangle_13" at 78,171 size 6x39
      Appearance <- "02_Peripheral_IN.AsitTahliyeVanasi.Opened"
   Rectangle "Rectangle_14" at 161,171 size 6x39
      Appearance <- "02_Peripheral_IN.AsitTahliyeVanasi.Closed"
   Rectangle "Rectangle_15" at 247,27 size 6x39
      Appearance <- "02_Peripheral_IN.UcYolluVana.Opened"
   Rectangle "Rectangle_16" at 328,27 size 6x39
      Appearance <- "02_Peripheral_IN.UcYolluVana.Closed"
   Rectangle "Rectangle_17" at 247,97 size 6x39
      Appearance <- "02_Peripheral_IN.KuyuAktVanasi.Opened"
   Rectangle "Rectangle_18" at 328,97 size 6x39
      Appearance <- "02_Peripheral_IN.KuyuAktVanasi.Closed"
   Rectangle "Rectangle_19" at 246,171 size 6x39
      Appearance <- "02_Peripheral_IN.IBC.AkisValfi.Opened"
   Rectangle "Rectangle_20" at 327,171 size 6x39
      Appearance <- "02_Peripheral_IN.IBC.AkisValfi.Closed"
   Rectangle "Rectangle_21" at 459,26 size 6x39
      Appearance <- "02_Peripheral_OUT.SuDolumVanasi"
   Rectangle "Rectangle_22" at 459,67 size 6x39
      Appearance <- "02_Peripheral_OUT.SuDolumVanasi"

screen "02_Alarm" 480x272, template "00_RootTamplate"
   AlarmView "Alarm view_1" at 0,0 size 479x222

screen "03_Izleme" 480x272, template "00_RootTamplate"
   TextField "Text field_1" at 11,23 size 68x28; Text 'Sirkulasyon Vanası'
   Circle "Circle_1" at 101,25 size 28x28
      Appearance <- "02_Peripheral_IN.SirkulasyonVanasi.Opened"
   Circle "Circle_2" at 142,25 size 28x28
      Appearance <- "02_Peripheral_IN.SirkulasyonVanasi.Closed"
   TextField "Text field_2" at 101,1 size 29x18; Text 'Açık'
   TextField "Text field_3" at 138,1 size 40x18; Text 'Kapalı'
   TextField "Text field_4" at 28,55 size 39x28; Text 'Dolum Vanası'
   Circle "Circle_3" at 101,57 size 28x28
      Appearance <- "02_Peripheral_IN.DolumVanasi.Opened"
   Circle "Circle_4" at 142,56 size 28x28
      Appearance <- "02_Peripheral_IN.DolumVanasi.Closed"
   TextField "Text field_5" at 11,87 size 68x28; Text 'Asit Tahliye Vanası'
   Circle "Circle_5" at 101,88 size 28x28
      Appearance <- "02_Peripheral_IN.AsitTahliyeVanasi.Opened"
   Circle "Circle_6" at 142,88 size 28x28
      Appearance <- "02_Peripheral_IN.AsitTahliyeVanasi.Closed"
   TextField "Text field_6" at 21,120 size 49x28; Text 'Uc Yollu Vana'
   Circle "Circle_7" at 101,120 size 28x28
      Appearance <- "02_Peripheral_IN.UcYolluVana.Opened"
   Circle "Circle_8" at 142,120 size 28x28
      Appearance <- "02_Peripheral_IN.UcYolluVana.Closed"
   TextField "Text field_7" at 11,151 size 74x28; Text 'Kuyu Tahliye Vanası'
   Circle "Circle_9" at 101,152 size 28x28
      Appearance <- "02_Peripheral_IN.KuyuAktVanasi.Opened"
   Circle "Circle_10" at 142,152 size 28x28
      Appearance <- "02_Peripheral_IN.KuyuAktVanasi.Closed"
   TextField "Text field_9" at 282,1 size 29x18; Text 'Açık'
   TextField "Text field_10" at 319,1 size 40x18; Text 'Kapalı'
   TextField "Text field_12" at 190,23 size 78x28; Text 'Yıkama Tankı Kapı Sw 1'
   Circle "Circle_15" at 283,23 size 28x28
      Appearance <- "02_Peripheral_IN.YikamaTanki.KapiSwitch1"
   Circle "Circle_16" at 324,23 size 28x28
      Appearance <- "02_Peripheral_IN.YikamaTanki.KapiSwitch1"
   TextField "Text field_14" at 194,54 size 58x28; Text 'Asit Tankı Kapı Sw'
   Circle "Circle_19" at 283,54 size 28x28
      Appearance <- "02_Peripheral_IN.AsitTanki.KapiSwitch"
   Circle "Circle_20" at 324,54 size 28x28
      Appearance <- "02_Peripheral_IN.AsitTanki.KapiSwitch"
   TextField "Text field_15" at 381,5 size 75x18; Text 'Ana Pompa'
   Circle "Circle_21" at 400,28 size 34x34
      Appearance <- "02_Peripheral_OUT.AnaPompa"
   TextField "Text field_16" at 381,72 size 80x18; Text 'IBC Pompası'
   Circle "Circle_22" at 399,97 size 34x34
      Appearance <- "02_Peripheral_OUT.IBC.PompaDiyafram"
   TextField "Text field_11" at 386,142 size 64x34; Text 'Kör Kuyu Pompası'
   Circle "Circle_13" at 399,178 size 34x34
      Appearance <- "02_Peripheral_OUT.KorKuyuPompasi"
   TextField "Text field_13" at 10,183 size 69x30; Text 'IBC Tahliye Vanası'
   Circle "Circle_14" at 100,185 size 28x28
      Appearance <- "02_Peripheral_IN.IBC.AkisValfi.Opened"
   Circle "Circle_17" at 141,185 size 28x28
      Appearance <- "02_Peripheral_IN.IBC.AkisValfi.Closed"
   TextField "Text field_8" at 287,88 size 21x18; Text 'Alt'
   TextField "Text field_17" at 327,88 size 23x18; Text 'Üst'
   TextField "Text field_18" at 197,169 size 61x41; Text 'Asti Tankı Seviye Alt/Üst'
   TextField "Text field_19" at 190,115 size 81x41; Text 'Yıkama Tankı Seviye Alt/Üst'
   Circle "Circle_11" at 279,121 size 34x34
      Appearance <- "02_Peripheral_IN.YikamaTanki.AltSeviyeSen"
   Circle "Circle_12" at 320,121 size 34x34
      Appearance <- "02_Peripheral_IN.YikamaTanki.UstSeviyeSen"
   Circle "Circle_18" at 279,174 size 34x34
      Appearance <- "02_Peripheral_IN.AsitTanki.AltSeviyeSen"
   Circle "Circle_23" at 320,174 size 34x34
      Appearance <- "02_Peripheral_IN.AsitTanki.UstSeviyeSen"

screen "04_Sure" 480x272, template "00_RootTamplate"
   IOField "I/O field_1" at 244,95 size 175x40; FormatPattern 9999999999; Unit  dk
      ProcessValue <- "03_HmiData_TimerInterval.AsitSirkulasyon"
   TextField "Text field_1" at 45,104 size 187x20; Text 'Asit Sirkülasyon Zamanı:'
   IOField "I/O field_2" at 244,150 size 176x40; FormatPattern 9999999999; Unit  dk
      ProcessValue <- "03_HmiData_TimerInterval.SuSirkulasyon"
   TextField "Text field_2" at 45,161 size 177x20; Text 'Su Sirkülasyon Zamanı:'
   Rectangle "Rectangle_1" at 26,7 size 419x57
      Visibility <- "03_HmiData_Visualization.TimerVisible"
   IOField "I/O field_3" at 138,37 size 107x24; FormatPattern 99999; Unit  dk
      Visibility <- "03_HmiData_Visualization.TimerVisible"
      ProcessValue <- "03_HmiData_Visualization.ActTimer"
   TextField "Text field_3" at 194,8 size 92x20; Text 'Geçen Sure:'
      Visibility <- "03_HmiData_Visualization.TimerVisible"
   IOField "I/O field_4" at 240,37 size 84x24; FormatPattern 99; Unit  sn
      ProcessValue <- "03_HmiData_Visualization.ActTimerSec"
      Visibility <- "03_HmiData_Visualization.TimerVisible"

screen "00_Root screen_1" 480x272, template "00_RootTamplate"
   IOField "Template_I/O field_1" at 161,2 size 237x44; FormatPattern ??????????????????????????????????????????????????
      ProcessValue <- "01_System_SystemInfo"
   Rectangle "Rectangle_1" at 334,168 size 139x48
      Visibility <- "03_HmiData_Visualization.TimerVisible"
   DateTimeField "HmiScreenItemData" at 393,23 size 85x22
   DateTimeField "HmiScreenItemData_1" at 393,1 size 85x22
   Button "Button_9" at 5,6 size 145x49; TextOn 'MANUEL'; TextOff 'NORMAL'; TextList "TextList_Manuel_Normal"
      on Release: InvertBit("01_System_Process.Manuel_Normal")
      Appearance <- "01_System_Process.Manuel_Normal"
      ProcessValue <- "01_System_Process.Manuel_Normal"
   Button "Button_15" at 5,59 size 145x49; TextOff 'Asit Doldur Başlat'
      on Press: function_b14e0dd5("03_HmiData_System.AsitDoldurBaslat", 0)
      Appearance <- "03_HmiData_Started.AsitDolum"
   Button "Button_1" at 174,54 size 135x50; TextOff 'Asit Sirkülasyon Başlat'
      on Press: function_b14e0dd5("03_HmiData_System.AsitSirkulasyonBaslat", 0)
      Appearance <- "03_HmiData_Started.AsitSirkulasyon"
   Button "Button_2" at 334,54 size 138x50; TextOff 'Asit Tahliyesi Başlat'
      on Press: function_b14e0dd5("03_HmiData_System.AsitTahliyesiBaslat", 0)
      Appearance <- "03_HmiData_Started.AsitTahliye"
   Button "Button_3" at 5,114 size 145x49; TextOff 'Su Dolum Başlat'
      on Press: function_b14e0dd5("03_HmiData_System.TemizSuDolumuBaslat", 0)
      Appearance <- "03_HmiData_Started.TemizSuDolum"
   Button "Button_4" at 174,112 size 135x50; TextOff 'Su Sirkülasyon Başlat'
      on Press: function_b14e0dd5("03_HmiData_System.TemizSuSirkulasyonuBaslat", 0)
      Appearance <- "03_HmiData_Started.TemizSuSirkulasyon"
   Button "Button_5" at 334,112 size 138x50; TextOff 'Su Tahliyesi Başlat'
      on Press: function_b14e0dd5("03_HmiData_System.TemizSuTahliyesiBaslat", 0)
      Appearance <- "03_HmiData_Started.TemizSuTahliye"
   Button "Button_6" at 5,168 size 146x49; TextOff 'IBC Tahliye Başlat'
      on Press: function_b14e0dd5("03_HmiData_System.IBCTahliyesiBaslat", 0)
      Appearance <- "03_HmiData_Started.IBCTahliye"
   Button "Button_7" at 246,168 size 83x49; TextOff 'Uyarı Sustur'
      on Press: function_b14e0dd5("03_HmiData_System.WarningReset", 0)
   Button "Button_8" at 157,168 size 83x49; TextOff 'İşlemi Durdur'
      on Press: function_b14e0dd5("03_HmiData_System.Stop", 0)
   IOField "I/O field_1" at 335,190 size 80x24; FormatPattern 9999; Unit  dk
      Visibility <- "03_HmiData_Visualization.TimerVisible"
      ProcessValue <- "03_HmiData_Visualization.ActTimer"
   TextField "Text field_1" at 365,168 size 80x18; Text 'Geçen Sure:'
      Visibility <- "03_HmiData_Visualization.TimerVisible"
   IOField "I/O field_2" at 414,190 size 58x24; FormatPattern 99; Unit  sn
      ProcessValue <- "03_HmiData_Visualization.ActTimerSec"
      Visibility <- "03_HmiData_Visualization.TimerVisible"

screen "01_Manuel_1" 480x272, template "00_RootTamplate"
   Button "Button_1" at 7,27 size 74x39; TextOff 'Ac'
      on Release: InvertBit("03_HmiData_SurkilasyonVanasi_Ac")
      Appearance <- "03_HmiData_SurkilasyonVanasi_Ac"
   Button "Button_2" at 9,97 size 74x39; TextOff 'Ac'
      on Release: InvertBit("03_HmiData_DolumVanasi_Ac")
      Visibility <- "03_HmiData_Visualization.Visibility.Manuel.DolumVanaAc"
      Appearance <- "03_HmiData_DolumVanasi_Ac"
   Button "Button_3" at 179,27 size 74x39; TextOff 'Ac'
      on Release: InvertBit("03_HmiData_UcYolluVana_Ac")
      Visibility <- "03_HmiData_Visualization.Visibility.Manuel.UcYolluVanaAc"
      Appearance <- "03_HmiData_UcYolluVana_Ac"
   Button "Button_5" at 179,97 size 74x39; TextOff 'Ac'
      on Release: InvertBit("03_HmiData_KuyuAktarimVanasi_Ac")
      Visibility <- "03_HmiData_Visualization.Visibility.Manuel.KuyuTahVanaAc"
      Appearance <- "03_HmiData_KuyuAktarimVanasi_Ac"
   Button "Button_4" at 8,171 size 74x39; TextOff 'Ac'
      on Release: InvertBit("03_HmiData_AsitTahliyeVanasi_Ac")
      Visibility <- "03_HmiData_Visualization.Visibility.Manuel.AsitTahVanaAc"
      Appearance <- "03_HmiData_AsitTahliyeVanasi_Ac"
   Button "Button_6" at 179,171 size 74x39; TextOff 'Ac'
      on Release: InvertBit("03_HmiData_IBCVanasi_Ac")
      Visibility <- "03_HmiData_Visualization.Visibility.Manuel.IBCVanaAc"
      Appearance <- "03_HmiData_IBCVanasi_Ac"
   Button "Button_7" at 346,67 size 117x39; TextOff 'Durdur'
      on Press: function_b14e0dd5("03_HmiData_AnaPompa_Stop", 0)
   Button "Button_8" at 345,169 size 119x39; TextOff 'Durdur'
      on Press: function_b14e0dd5("03_HmiData_IBC_DiyaframPompa_Stop", 0)
   Button "Button_9" at 89,27 size 74x39; TextOff 'Kapat'
      on Release: InvertBit("03_HmiData_SurkilasyonVanasi_Kapat")
      Appearance <- "03_HmiData_SurkilasyonVanasi_Kapat"
   Button "Button_10" at 258,27 size 74x39; TextOff 'Kapat'
      on Release: InvertBit("03_HmiData_UcYolluVana_Kapat")
      Visibility <- "03_HmiData_Visualization.Visibility.Manuel.UcYolluVanaKapat"
      Appearance <- "03_HmiData_UcYolluVana_Kapat"
   Button "Button_11" at 89,97 size 74x39; TextOff 'Kapat'
      on Release: InvertBit("03_HmiData_DolumVanasi_Kapat")
      Visibility <- "03_HmiData_Visualization.Visibility.Manuel.DolumVanaKapat"
      Appearance <- "03_HmiData_DolumVanasi_Kapat"
   Button "Button_12" at 87,171 size 74x39; TextOff 'Kapat'
      on Release: InvertBit("03_HmiData_AsitTahliyeVanasi_Kapat")
      Visibility <- "03_HmiData_Visualization.Visibility.Manuel.AsitTahVanaKapat"
      Appearance <- "03_HmiData_AsitTahliyeVanasi_Kapat"
   Button "Button_13" at 258,97 size 74x39; TextOff 'Kapat'
      on Release: InvertBit("03_HmiData_KuyuAktarimVanasi_Kapat")
      Visibility <- "03_HmiData_Visualization.Visibility.Manuel.KuyuTahVanaKapat"
      Appearance <- "03_HmiData_KuyuAktarimVanasi_Kapat"
   Button "Button_14" at 258,171 size 74x39; TextOff 'Kapat'
      on Release: InvertBit("03_HmiData_IBCVanasi_Kapat")
      Visibility <- "03_HmiData_Visualization.Visibility.Manuel.IBCVanaKapat"
      Appearance <- "03_HmiData_IBCVanasi_Kapat"
   Button "Button_15" at 346,24 size 117x39; TextOff 'Çalıştır'
      on Press: function_b14e0dd5("03_HmiData_AnaPompa_Run", 0)
      Appearance <- "HmiAnaPompa_Run"
   Button "Button_16" at 344,126 size 119x39; TextOff 'Çalıştır'
      on Press: function_b14e0dd5("03_HmiData_IBC_DiyaframPompa_Run", 0)
      Appearance <- "HmiIBCPopmpa_Run"
   TextField "Text field_1" at 25,5 size 123x18; Text 'Sirkülasyon Vanasi'
   TextField "Text field_3" at 39,78 size 88x18; Text 'Dolum Vanasi'
   TextField "Text field_4" at 21,149 size 124x18; Text 'Asit Tahliye Vanasi'
   TextField "Text field_5" at 214,5 size 89x18; Text 'Uc Yollu Vana'
   TextField "Text field_6" at 185,78 size 136x18; Text 'Kuyu Aktarım Vanası'
   TextField "Text field_7" at 216,150 size 70x18; Text 'IBC Vanasi'
   TextField "Text field_2" at 366,5 size 75x18; Text 'Ana Pompa'
   TextField "Text field_8" at 369,108 size 70x18; Text 'IBC Pompa'

screen "01_Manuel_Syf2" 480x272
   TextField "Text field_2" at 204,7 size 75x18; Text 'Ana Pompa'
   TextField "Text field_8" at 204,95 size 70x18; Text 'IBC Pompa'
   TextField "Text field_1" at 184,186 size 117x18; Text 'Kör Kuyu Pompası'
   Button "Button_3" at 8,183 size 53x85; TextOff 'Text'; PictureOff "Left_Arrow"
      on Release: ActivateScreen("01_Manuel", 0)
   Button "Button_7" at 253,32 size 117x39; TextOff 'Durdur'
      on Press: function_b14e0dd5("03_HmiData_AnaPompa_Stop", 0)
   Button "Button_8" at 253,120 size 119x39; TextOff 'Durdur'
      on Press: function_b14e0dd5("03_HmiData_IBC_DiyaframPompa_Stop", 0)
   Button "Button_15" at 112,32 size 117x39; TextOff 'Çalıştır'
      on Press: function_b14e0dd5("03_HmiData_AnaPompa_Run", 0)
      Appearance <- "HmiAnaPompa_Run"
   Button "Button_16" at 112,121 size 119x39; TextOff 'Çalıştır'
      on Press: function_b14e0dd5("03_HmiData_IBC_DiyaframPompa_Run", 0)
      Appearance <- "HmiIBCPopmpa_Run"
   Button "Button_1" at 253,210 size 119x39; TextOff 'Durdur'
      on Press: function_b14e0dd5("03_HmiData_KorKuyuPompası_Stop", 0)
   Button "Button_2" at 112,210 size 119x39; TextOff 'Çalıştır'
      on Press: function_b14e0dd5("03_HmiData_KorKuyuPompası_Run", 0)
      Appearance <- "HmiKorKuyuPompa_Run"
*)